TEXTLIST textListLeft
  0 = ''
  1 = 'X'
  2 = '>'
  3 = '<'
   = ''
END_TEXTLIST

(* stored: Version 1.1.0.1, ProductVersion 3.1.4024.11
   TextList textListLeft: Id {c444fabb-59aa-089e-157d-acff22ede57f} *)
